PROGRAM MC_State_MC
VAR
END_VAR

//fbMC_Home.Options.ClearPositionLag := TRUE;
//fbMC_Home.Options.ReferenceMode;
//fbMC_Home.Options.SearchDirection;
//fbMC_Home.Options.SearchVelocity;
//fbMC_Home.Options.SyncDirection;
//fbMC_Home.Options.SyncVelocity;


Act_MotionAbsolute();
Act_MotionHome();
Act_MotionManual();
Act_MotionPower();
Act_MotionReset();

ACTION Act_MotionAbsolute:
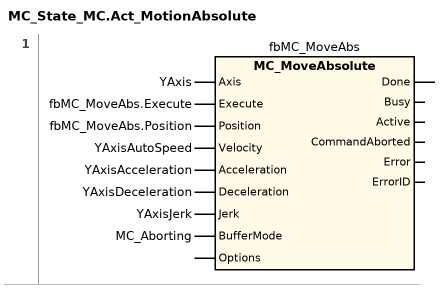
// NETWORK 1
fbMC_MoveAbs(
    Axis := YAxis,
    Execute := fbMC_MoveAbs.Execute,
    Position := fbMC_MoveAbs.Position,
    Velocity := YAxisAutoSpeed,
    Acceleration := YAxisAcceleration,
    Deceleration := YAxisDeceleration,
    Jerk := YAxisJerk,
    BufferMode := MC_Aborting); // MC_MoveAbsolute
END_ACTION

ACTION Act_MotionHome:
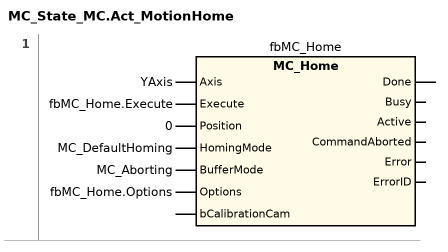
// NETWORK 1
fbMC_Home(
    Axis := YAxis,
    Execute := fbMC_Home.Execute,
    Position := 0,
    HomingMode := MC_DefaultHoming,
    BufferMode := MC_Aborting,
    Options := fbMC_Home.Options); // MC_Home
END_ACTION

ACTION Act_MotionManual:
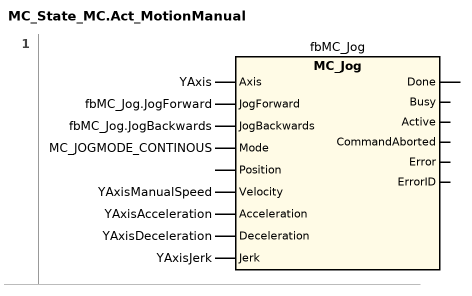
// NETWORK 1
fbMC_Jog(
    Axis := YAxis,
    JogForward := fbMC_Jog.JogForward,
    JogBackwards := fbMC_Jog.JogBackwards,
    Mode := MC_JOGMODE_CONTINOUS,
    Velocity := YAxisManualSpeed,
    Acceleration := YAxisAcceleration,
    Deceleration := YAxisDeceleration,
    Jerk := YAxisJerk); // MC_Jog
END_ACTION

ACTION Act_MotionPower:
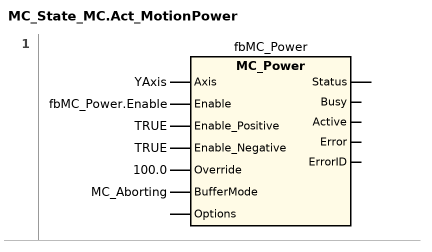
// NETWORK 1
fbMC_Power(
    Axis := YAxis,
    Enable := fbMC_Power.Enable,
    Enable_Positive := TRUE,
    Enable_Negative := TRUE,
    Override := 100.0,
    BufferMode := MC_Aborting); // MC_Power
END_ACTION

ACTION Act_MotionReset:
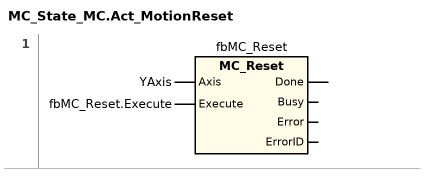
// NETWORK 1
fbMC_Reset(Axis := YAxis, Execute := fbMC_Reset.Execute); // MC_Reset
END_ACTION

END_PROGRAM

(* stored: Version 1.1.0.1, ProductVersion 3.1.4024.3
   POU MC_State_MC: Id {120a86f4-9f67-4bdd-9249-5865d99ceb30}, SpecialFunc None
   Action Act_MotionAbsolute: Id {e963b8a7-70b5-4b37-92e5-ca50e1d6823d}
   Action Act_MotionHome: Id {72103340-1220-4962-a7e8-eb5f2b1603a7}
   Action Act_MotionManual: Id {fc54c6e1-b939-4e3c-aaaf-8584342dc070}
   Action Act_MotionPower: Id {119c7967-2b0f-45aa-8596-148e8e07b830}
   Action Act_MotionReset: Id {53dcda7e-c948-49fd-a7f8-723398cb1136} *)
